// TIA Portal V21 export
DATA_BLOCK "Ao_Faceplate_Db"   // DB105
{ S7_Optimized_Access := 'FALSE' }
// stored: AutoNumber false
   VAR
      Mm01Ref : "Ao_Faceplate";
      Cp01Ref : "Ao_Faceplate";
      Cv01 : "Ao_Faceplate";
      AoSpare1 : "Ao_Faceplate";
      AoSpare2 : "Ao_Faceplate";
      AoSpare3 : "Ao_Faceplate";
      AoSpare4 : "Ao_Faceplate";
      AoSpare5 : "Ao_Faceplate";
   END_VAR
BEGIN
END_DATA_BLOCK
